// TIA Portal V17 export
// export: Created 2025-03-05T08:01:20.4596974Z, ExportSetting WithDefaults, DisplayName Totally Integrated Automation Portal, DisplayVersion V17 Update 8, DisplayName TIA Portal Openness, DisplayVersion V17 Update 8, DisplayName TIA Portal Version Control Interface, DisplayVersion V17, DisplayName SINAMICS Startdrive Advanced, DisplayVersion V17 SP2, DisplayName SINAMICS Startdrive G110M, G120, G120C, G120D, G120P, G115D, DisplayVersion V17 SP2, DisplayName SINAMICS Startdrive G130, G150, S120, S150, SINAMICS MV, S210, DisplayVersion V17 SP2, DisplayName STEP 7 Professional, DisplayVersion V17 Update 8, DisplayName SINUMERIK ONE STEP 7 Toolbox, DisplayVersion V17 Update 12, DisplayName SINUMERIK 840D sl STEP 7 Toolbox, DisplayVersion V17 Update 12, DisplayName STEP 7 Safety, DisplayVersion V17 Update 6, DisplayName WinCC Advanced, DisplayVersion V17 Update 8
DATA_BLOCK "DB6892_SAFETY_BRAKE_AXIS_Z23"   // DB6892
{ DB_Accessible_From_OPC_UA := 'FALSE' }
AUTHOR : ETXETAR
VERSION : 1.0
// stored: AutoNumber false, DBAccessibleFromOPCUA false, DBAccessibleFromWebserver true, InstanceOfName FB6600_SAFETY_BRAKE_Z_AXIS, InstanceOfType FB
"FB6600_SAFETY_BRAKE_Z_AXIS"
   // VAR_INPUT
   //    OPTIONS_0 : Byte;
   //    BLOCKED_1 : Bool;
   //    UNBLOCKED_1 : Bool;
   //    MAINT_BLOCKED : Bool;
   //    MAINT_UNBLOCKED : Bool;
   //    BLOCK_CONDITIONS : Bool;
   //    UNBLOCK_CONDITIONS : Bool;
   //    AXIS_SELECTED : Bool;
   //    TRAVERSE_COMMAND : Bool;
   //    UNBLOCK_MAN_REQUEST : Bool;
   //    BLOCK_AUTO_REQUEST : Bool;
   //    UNBLOCK_AUTO_REQUEST : Bool;
   //    BRAKE_TEST : Bool;
   //    UNIT_ALARM : UInt;
   //    STATION_ALARM : UInt;
   // END_VAR
   // VAR_OUTPUT
   //    BLOCKED : Bool;
   //    UNBLOCKED : Bool;
   //    BLOCKED_ALARM : Bool;
   //    UNBLOCKED_ALARM : Bool;
   //    MAINTENANCE_UNBLOCKED_ALARM : Bool;
   //    BLOCK : Bool;
   //    UNBLOCK : Bool;
   // END_VAR
   // VAR RETAIN
   //    BRAKE { S7_SetPoint := 'True'} : "SAFETY_BRAKE";
   //    TIMER_BLOCKED { S7_SetPoint := 'True'} : TON_TIME;
   //    TIMER_UNBLOCKED { S7_SetPoint := 'True'} : TON_TIME;
   //    TIMER_SIMULTANEITY { S7_SetPoint := 'True'} : TON_TIME;
   //    TIMER_TIME_EXCEEDED { S7_SetPoint := 'True'} : TON_TIME;
   // END_VAR
BEGIN
END_DATA_BLOCK
